FUNCTION_BLOCK FB_No_start
VAR_INPUT
	Run:BOOL;
	No_start_trip:BOOL;
	Reset:BOOL;
	Run_FB:BOOL;
	CB_trip:BOOL;
	CB_On:BOOL;
	Use_int_estop:BOOL; (*Internally generated E-Stop when Contactor feedback is lost without removing run command*)
	Ext_estop:BOOL; (*External Estop with monitored contact*)
	Ns_time:TIME;
END_VAR
VAR_OUTPUT
	NS_trip:BOOL;
	Estop_out:BOOL;
END_VAR
VAR
	TON_0: TON;
	SR_0: SR;
	F_TRIG_0: F_TRIG;
	SR_1: SR;
END_VAR

M_Main();

METHOD M_Main
VAR_INPUT
END_VAR
VAR_INST // added by the converter: edge detectors and wires of the graphical bodies
    _w1, _w3, _w4 : BOOL;
    _w2 : ANY;
END_VAR
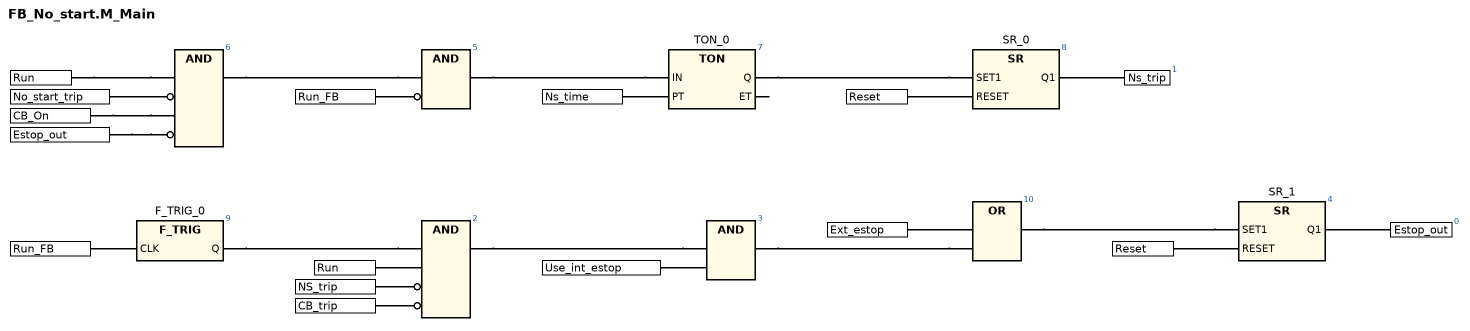
Estop_out := SR_1.Q1;
Ns_trip := SR_0.Q1;
_w1 := (F_TRIG_0.Q AND Run AND NOT NS_trip AND NOT CB_trip) AND Use_int_estop;
SR_1(SET1 := _w2, RESET := Reset); // SR
_w4 := _w3 AND NOT Run_FB;
_w3 := Run AND NOT No_start_trip AND CB_On AND NOT Estop_out;
TON_0(IN := _w4, PT := Ns_time); // TON
SR_0(SET1 := TON_0.Q, RESET := Reset); // SR
F_TRIG_0(CLK := Run_FB); // F_TRIG
_w2 := Ext_estop OR _w1;
END_METHOD

END_FUNCTION_BLOCK

(* stored: Version 1.1.0.1, ProductVersion 3.1.4024.0
   POU FB_No_start: Id {65fec9db-edad-4c28-b5dd-8e5c9a4e9ba8}, SpecialFunc None
   Method M_Main: Id {f949ef21-8f17-428f-80ce-287468964702} *)
